TYPE Array8_LReal :
UNION
	arrByte			:ARRAY[0..7] OF BYTE;
	rValue			:LREAL;
END_UNION
END_TYPE

(* stored: Version 1.1.0.1
   DUT Array8_LReal: Id {a272c096-0205-4fda-8871-e23133a7cb7f} *)
